TYPE UNI_HMI_WheelHouseInput :
UNION
	arWheelHouseInput : ARRAY[1..400] OF BOOL;
	List :ST_WheelhouseInput;
END_UNION
END_TYPE

(* stored: Version 1.1.0.1, ProductVersion 3.1.4024.13
   DUT UNI_HMI_WheelHouseInput: Id {3e7e253c-da37-415f-8ad6-d848888beba2} *)
